ABB RobotStudio station: sesion6_EstacionDePartidaSoloRobotFin.rspag

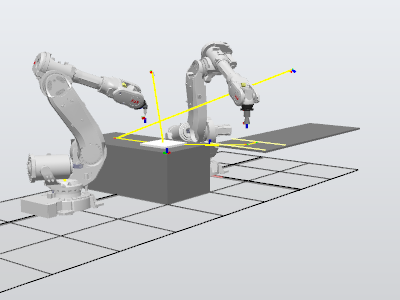
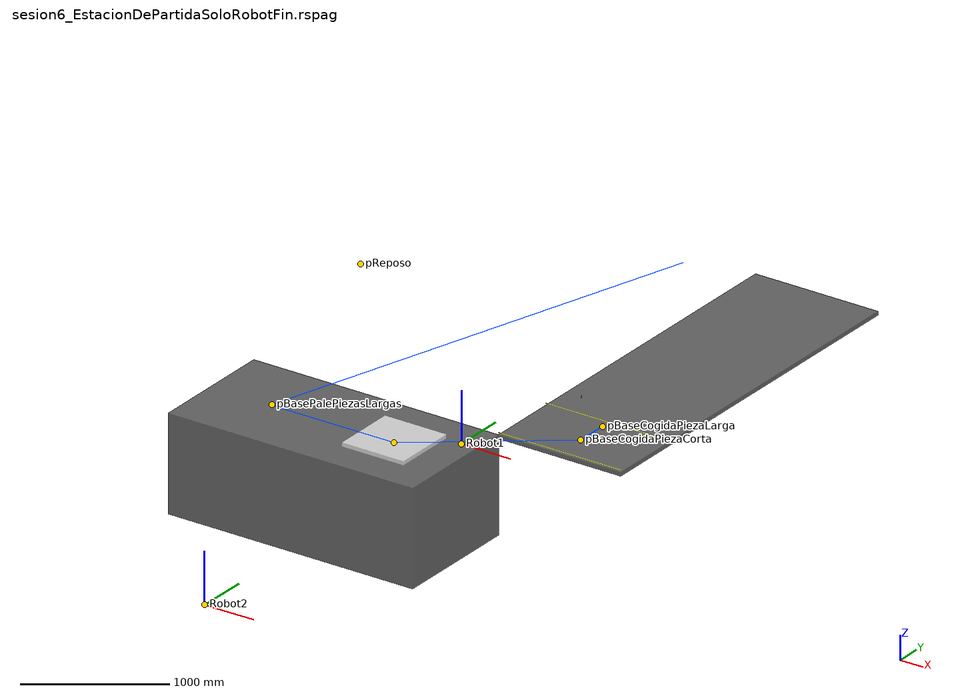
[picture v1: parts stored in the station drawn from their meshes, with robot base, taught points and paths (robot models come from the ABB library and are not in the file)]
--- station ---
Station sesion7_EstacionDePartida_1 (saved by RobotStudio 24.1.10713.1)
Controller Controlador3, task T_ROB1: task frame (RAPID world) sits at (0, -3000, 0) mm, rotated rx 0 ry 0 rz 90 deg in the station
Controller Sistema6
  mechanical unit ROB_1: Robot1, 6 joints, base frame (0, 0, 0) mm
Controller Controlador3
  mechanical unit ROB_1: Robot2, 6 joints, base frame (0, 0, 0) mm
Layout (positions relative to the parent item):
  - Ventosa [mechanism] at (1500, -750, 1280) mm, rotated rx -180 ry 0 rz -180 deg
      TCP Ventosa at (0, 0, 200) mm
      links: PiezaVentosa
  - Robot1 [mechanism, from %ABB.RobotStudio.Models.IRB6640%\IRB6640_180_255_G_04.rslib] at (0, 0, 0) mm; joint values [-0.4636, 0.2346, 0.2413, 0, 1.095, -0.4636] (rad or m)
  - CI_VentosaVacuostato [smart component]
      signals: DI ActivaVentosa, DO Vacuostato
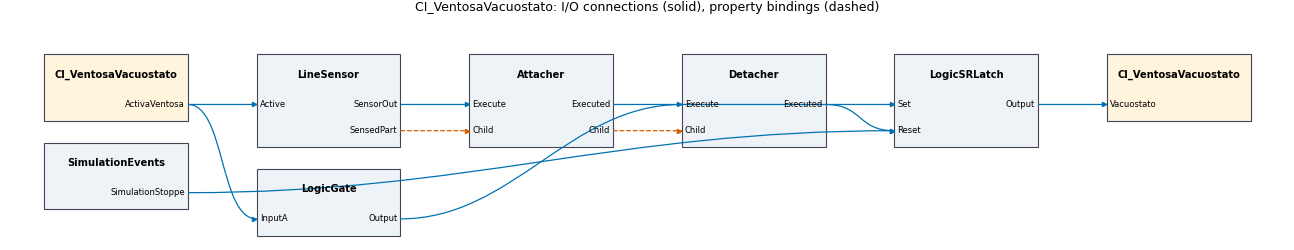
      connections:
        CI_VentosaVacuostato.ActivaVentosa -> LineSensor.Active
        LineSensor.SensorOut -> Attacher.Execute
        Attacher.Executed -> LogicSRLatch.Set
        LogicSRLatch.Output -> CI_VentosaVacuostato.Vacuostato
        Detacher.Executed -> LogicSRLatch.Reset
        SimulationEvents.SimulationStopped -> LogicSRLatch.Reset
        CI_VentosaVacuostato.ActivaVentosa -> LogicGate.InputA
        LogicGate.Output -> Detacher.Execute
        LineSensor.SensedPart => Attacher.Child
        Attacher.Child => Detacher.Child
    - LineSensor [smart component, from Components\LineSensor.rslib] at (1500, -750, 1080) mm, rotated rx -180 ry 0 rz -180 deg
        properties: Start=[0 0 -0.002]; End=[0 0 0.02]; Radius=0.002; SensedPart=(none); SensedPoint=[0.5 -1.49999987792969 0.780095153808594]; Length=0.022; Tag=(none)
      - _sensorPart_ [part], size 4 x 4 x 22 mm
    - SimulationEvents [smart component, from Components\SimulationEvents.rslib]
    - LogicSRLatch [smart component, from Components\LogicSRLatch.rslib]
    - Attacher [smart component, from Components\Attacher.rslib]
        properties: Parent=Ventosa; Flange=0; Child=(none); Mount=false; Offset=[0 0 0]; Orientation=[0 0 0]
    - Detacher [smart component, from Components\Detacher.rslib]
        properties: Child=(none); KeepPosition=true
    - LogicGate [smart component, from Components\LogicGate.rslib]
        properties: Operator=NOT; Delay=0.1
  - MesaPaletizadoParteIzq [part], size 1000 x 1000 x 750 mm
  - MesaPaletizadoParteDer [part], size 1000 x 1000 x 750 mm
  - cintaTransportadora [part], size 1000 x 3000 x 30 mm
  - PiezaLarga [part], size 500 x 1000 x 30 mm
  - PiezaCorta [part], size 500 x 500 x 30 mm
  - CI_SensoresCinta [smart component]
      signals: DI ActivaSensores, DO FinalCintaDetectado, DO PiezaLargaDetectada
      connections:
        CI_SensoresCinta.ActivaSensores -> LineSensorFinalCinta.Active
        CI_SensoresCinta.ActivaSensores -> LineSensorPiezaLarga.Active
        LineSensorPiezaLarga.SensorOut -> CI_SensoresCinta.PiezaLargaDetectada
        LineSensorFinalCinta.SensorOut -> CI_SensoresCinta.FinalCintaDetectado
    - LineSensorFinalCinta [smart component, from Components\LineSensor.rslib]
        properties: Start=[1 -1 0.765]; End=[2 -1 0.765]; Length=1; Radius=0.002; Tag=(none); SensedPart=(none); SensedPoint=[0 0 0]
      - _sensorPart_ [part], size 1000 x 4 x 4 mm
    - LineSensorPiezaLarga [smart component, from Components\LineSensor.rslib]
        properties: Start=[1 -0.45 0.765]; End=[2 -0.45 0.765]; Length=1; Radius=0.002; Tag=(none); SensedPart=(none); SensedPoint=[0 0 0]
      - _sensorPart_ [part], size 1000 x 4 x 4 mm
  - CI_CintaTransportadora [smart component]
      signals: DI PideNuevaPieza, DI MueveCinta, DI Desencolar
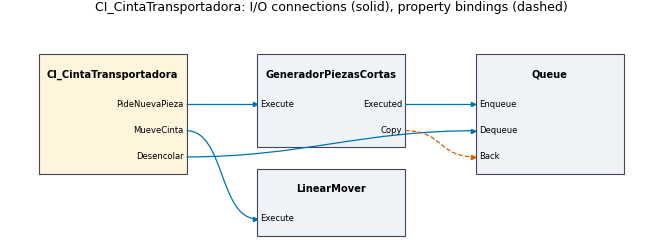
      connections:
        GeneradorPiezasCortas.Executed -> Queue.Enqueue
        CI_CintaTransportadora.PideNuevaPieza -> GeneradorPiezasCortas.Execute
        CI_CintaTransportadora.MueveCinta -> LinearMover.Execute
        CI_CintaTransportadora.Desencolar -> Queue.Dequeue
        GeneradorPiezasCortas.Copy => Queue.Back
    - GeneradorPiezasCortas [smart component, from Components\Source.rslib]
        properties: Source=PiezaCorta; Copy=(none); Parent=(none); Position=[1.25 1.5 0.75]; Orientation=[0 0 0]; Transient=false; PhysicsBehavior=-1
    - LinearMover [smart component, from Components\LinearMover.rslib]
        properties: Object=Queue; Direction=[0 -0.001 0]; Speed=0.2; Reference=Global; ReferenceObject=(none)
    - Queue [smart component, from Components\Queue.rslib]
        properties: Back=(none); Front=(none); Queue={d6de95e9-a5e4-462f-8fb5-12ca184cec83}; NumberOfObjects=0
  - PiezaCorta_5 [part] at (249.2, -1250, 750) mm, rotated rx 0 ry 0 rz -90 deg, size 500 x 500 x 30 mm
  - Robot2 [mechanism, from %ABB.RobotStudio.Models.IRB6640%\IRB6640_180_255_G_04.rslib] at (0, -3000, 0) mm, rotated rx 0 ry 0 rz 90 deg; joint values [-0.5264, -0.4516, 0.7886, 0.4989, 0.7029, -0.8234] (rad or m)
  - MyTool [mechanism, from Training Objects\myTool.rslib] at (500, -2016.33, 1400.53) mm, rotated rx 180 ry 38 rz -90 deg
Attachment: Ventosa is attached to Robot1 / Link6
Attachment: LineSensor is attached to Ventosa / PiezaVentosa
Attachment: MyTool is attached to Robot2 / Link6
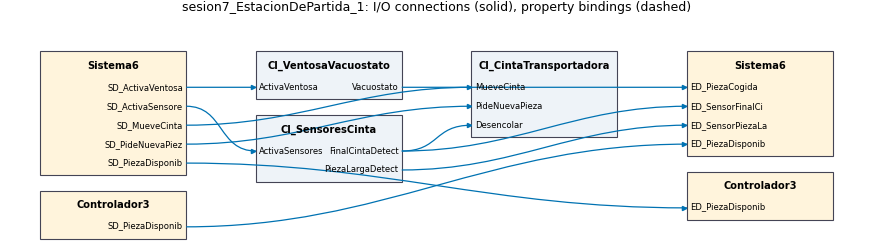
Station logic (signal -> signal, property => property):
  CI_VentosaVacuostato.Vacuostato -> Sistema6.ED_PiezaCogida
  Sistema6.SD_ActivaVentosa -> CI_VentosaVacuostato.ActivaVentosa
  CI_SensoresCinta.FinalCintaDetectado -> Sistema6.ED_SensorFinalCinta
  CI_SensoresCinta.PiezaLargaDetectada -> Sistema6.ED_SensorPiezaLarga
  Sistema6.SD_ActivaSensores -> CI_SensoresCinta.ActivaSensores
  Sistema6.SD_MueveCinta -> CI_CintaTransportadora.MueveCinta
  Sistema6.SD_PideNuevaPieza -> CI_CintaTransportadora.PideNuevaPieza
  CI_SensoresCinta.FinalCintaDetectado -> CI_CintaTransportadora.Desencolar
  Sistema6.SD_PiezaDisponible -> Controlador3.ED_PiezaDisponible
  Controlador3.SD_PiezaDisponibleAck -> Sistema6.ED_PiezaDisponibleAck

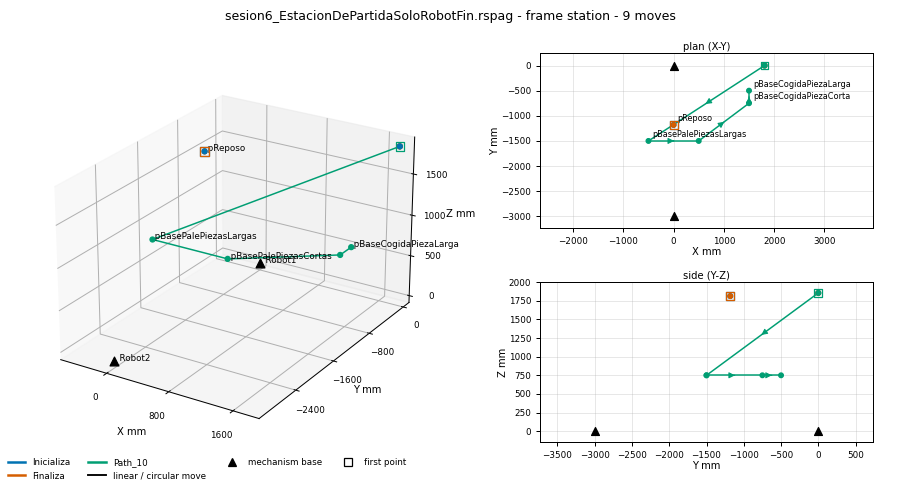
[picture p0: tool path of sesion6_EstacionDePartidaSoloRobotFin.rspag in frame station, 9 of 20 moves have a stored position in this frame; points joined in program order, loops and branches not executed]
--- Backups/Controlador3/RAPID/TASK1/PROGMOD/CalibData.mod ---
MODULE CalibData
    PERS tooldata MyTool:=[TRUE,[[31.792631019,0,229.638935148],[0.945518576,0,0.325568154,0]],[1,[0,0,1],[1,0,0,0],0,0,0]];
    TASK PERS wobjdata WO_Paletizado:=[FALSE,TRUE,"",[[1000,-1000,750],[1,0,0,0]],[[0,0,0],[1,0,0,0]]];
ENDMODULE

--- Backups/Controlador3/RAPID/TASK1/PROGMOD/Module1.mod ---
MODULE Module1
        CONST robtarget pReposo:=[[1818.681916784,0,1812.64730631],[0.190808996,0,0.981627183,0],[0,0,0,0],[9E+09,9E+09,9E+09,9E+09,9E+09,9E+09]];
    CONST robtarget pBasePalePiezasCortas:=[[500,500,0],[0,0,1,0],[-1,0,0,0],[9E+09,9E+09,9E+09,9E+09,9E+09,9E+09]];
    CONST robtarget pBasePalePiezasLargas:=[[500,1500,0],[0,0,1,0],[0,-1,0,0],[9E+09,9E+09,9E+09,9E+09,9E+09,9E+09]];
    PROC Inicializa ()
      MoveJ pReposo, v3000, fine, MyTool;
      Reset SD_PiezaDisponibleAck;
   ENDPROC
   PROC Finaliza ()
      MoveJ pReposo, v3000, fine, MyTool;
      Reset SD_PiezaDisponibleAck;
   ENDPROC
      PROC Main ()
      VAR num nPiezas;

      Inicializa;

      FOR nPiezas FROM 1 TO 20 DO
         WaitDI ED_PiezaDisponible, 1;
         SetDO SD_PiezaDisponibleAck, 1;
         WaitTime 0.3;
         Reset SD_PiezaDisponibleAck;
         TaladraPieza pBasePalePiezasCortas, nPiezas, 30;
      ENDFOR

      Finaliza;
   ENDPROC
      PROC TaladraPieza (robtarget pBase, num nPiezas, num altoPieza)
      VAR robtarget pTaladrado;
      VAR robtarget pAprox;
      VAR robtarget pEspera;
      VAR num distSeguridadZ := 300;
      VAR num distSeguridadEsperaX := -400;


      pTaladrado := Offs (pBasePalePiezasCortas, 0, 0, altoPieza*nPiezas);
      pAprox := Offs (pTaladrado, 0, 0, distSeguridadZ);
      pEspera := Offs (pTaladrado, distSeguridadEsperaX, 0, distSeguridadZ);

      MoveJ pAprox, v3000, z100, MyTool, \WObj:=WO_Paletizado;
      MoveL pTaladrado, v1000, fine, MyTool, \WObj:=WO_Paletizado;
      ! Aquí accionaríamos taladro. Simulamos con espera de 0.3 segundos:
      WaitTime 0.3;
      MoveL pAprox, v1000, z100, MyTool, \WObj:=WO_Paletizado;
      MoveJ pEspera, v3000, z100, MyTool, \WObj:=WO_Paletizado;
   ENDPROC
ENDMODULE

--- Backups/Sistema6/RAPID/TASK1/PROGMOD/CalibData.mod ---
MODULE CalibData
	PERS tooldata Ventosa:=[TRUE,[[0,0,200],[1,0,0,0]],[1,[0,0,125],[1,0,0,0],0.002,0.002,0.0013]];
    TASK PERS wobjdata WO_Paletizado:=[FALSE,TRUE,"",[[1000,-2000,750],[0.707106781,0,0,0.707106781]],[[0,0,0],[1,0,0,0]]];
    TASK PERS wobjdata WO_CintaTransportadora:=[FALSE,TRUE,"",[[1000,-1000,750],[1,0,0,0]],[[0,0,0],[1,0,0,0]]];
ENDMODULE

--- Backups/Sistema6/RAPID/TASK1/PROGMOD/Module1.mod ---
MODULE Module1
    CONST robtarget pReposo:=[[1808.910161514,0,1855],[0.5,0,0.866025404,0],[0,0,0,0],[9E+09,9E+09,9E+09,9E+09,9E+09,9E+09]];
    CONST robtarget pBasePalePiezasLargas:=[[500,1500,0],[0,1,0,0],[-2,0,-1,0],[9E+09,9E+09,9E+09,9E+09,9E+09,9E+09]];
    CONST robtarget pBasePalePiezasCortas:=[[500,500,0],[0,1,0,0],[-1,0,0,0],[9E+09,9E+09,9E+09,9E+09,9E+09,9E+09]];
    CONST robtarget pBaseCogidaPiezaCorta:=[[500,250,0],[0,0,1,0],[-1,0,-1,0],[9E+09,9E+09,9E+09,9E+09,9E+09,9E+09]];
    CONST robtarget pBaseCogidaPiezaLarga:=[[500,500,0],[0,0,1,0],[-1,0,-1,0],[9E+09,9E+09,9E+09,9E+09,9E+09,9E+09]];
 PROC Inicializa ()
      MoveJ pReposo, v3000, fine, Ventosa, \WObj:=wobj0;
      Reset SD_ActivaVentosa;
      SetDO SD_ActivaSensores, 1;
      SetDO SD_MueveCinta, 1;
      Reset SD_PideNuevaPieza;
      Reset SD_PiezaDisponible;
   ENDPROC

   PROC Finaliza ()
      MoveJ pReposo, v3000, fine, Ventosa, \WObj:=wobj0;
      Reset SD_ActivaVentosa;
      Reset SD_PideNuevaPieza;
      Reset SD_MueveCinta;
      Reset SD_ActivaSensores;
      Reset SD_ActivaSensores;
      Reset SD_PiezaDisponible;
   ENDPROC

   PROC Main ()
      CONST num altoPieza := 30;
      VAR num nPiezas;

      Inicializa;

      FOR nPiezas FROM 1 TO 20 DO
         WaitDI ED_SensorFinalCinta, 1;
         LlevaPiezaAPale nPiezas, altoPieza;
         SetDO SD_PiezaDisponible, 1;
         WaitDI ED_PiezaDisponibleAck, 1;
         Reset SD_PiezaDisponible;
      ENDFOR

      Finaliza;
   ENDPROC

   PROC LlevaPiezaAPale (num nPiezas, num altoPieza)
      VAR robtarget pCoger;
      VAR robtarget pSoltar;
      VAR robtarget pCogerAprox;
      VAR robtarget pSoltarAprox;
      VAR num distSeguridad := 300;

      pCoger  := Offs (pBaseCogidaPiezaCorta, 0, 0, altoPieza);
      pSoltar := Offs (pBasePalePiezasCortas, 0, 0, altoPieza*nPiezas);

      pCogerAprox  := Offs (pCoger,  0, 0, distSeguridad);
      pSoltarAprox := Offs (pSoltar, 0, 0, distSeguridad);

      MoveJ pCogerAprox, v3000, z100, Ventosa, \WObj:=WO_CintaTransportadora;
      MoveLDO pCoger, v1000, fine, Ventosa, \WObj:=WO_CintaTransportadora, SD_ActivaVentosa, 1;
      WaitDI ED_PiezaCogida, 1;
      MoveL pCogerAprox, v1000, z100, Ventosa, \WObj:=WO_CintaTransportadora;
      MoveJ pSoltarAprox, v3000, z100, Ventosa, \WObj:=WO_Paletizado;
      MoveLDO pSoltar, v1000, fine, Ventosa, \WObj:=WO_Paletizado, SD_ActivaVentosa, 0;
      WaitDI ED_PiezaCogida, 0;
      MoveL pSoltarAprox, v1000, z100, Ventosa, \WObj:=WO_Paletizado;
      MoveJ pCogerAprox, v3000, z100, Ventosa, \WObj:=WO_CintaTransportadora;
   ENDPROC
    PROC Path_10()
        MoveL pReposo,v1000,z100,Ventosa\WObj:=wobj0;
        MoveL pBasePalePiezasLargas,v1000,z100,Ventosa\WObj:=WO_Paletizado;
        MoveL pBasePalePiezasCortas,v1000,z100,Ventosa\WObj:=WO_Paletizado;
        MoveL pBaseCogidaPiezaCorta,v1000,z100,Ventosa\WObj:=WO_CintaTransportadora;
        MoveL pBaseCogidaPiezaLarga,v1000,z100,Ventosa\WObj:=WO_CintaTransportadora;
    ENDPROC
ENDMODULE

--- Backups/Sistema6/RAPID/TASK1/SYSMOD/LINKEDM.sys ---
%%%
  VERSION:1
  LANGUAGE:ENGLISH
%%%

MODULE LINKEDM (SYSMODULE)

! FOLLOWER
!     Name of electronically linked follower axis used by operator at teach pendent.
      PERS string l_f_axis_name{5}       :=  ["",  "", "", "", ""];

!     Name of the mechanical unit for follower axis.
      PERS string l_f_mecunt_n{5}  :=  ["", "", "", "", ""];

!     Linked follower axis number in the mechanical unit (first axis in mech. unit is number 1).
      PERS num l_f_axis_no{5}      :=  [0,          0,   0,  0,  0];

! MASTER
!     Name of the mechanical unit for linked master axis.
      PERS string l_m_mecunt_n{5} :=  ["", "", "", "", ""];

!     Linked master axis number in the mechanical unit (first axis in mech. unit is number 1).
!     See axis number table in documentation for different master mechanical units.
      PERS num l_m_axis_no{5}     :=  [0,  0,  0,  0,  0];

! POSITION OFFSET
!     The increase of the allowed offset position between the master and follower
!     positions, used when starting AUTO mode. As soon as the offset is decreased
!     the old configurated parameter is used.
!     Example: 3 => the configurated value of allowed offset is increased 3 times.
      PERS num offset_ratio{5}       :=  [10,  10,   10,  10,  10];

! SPEED RATIO
!     Speed_ratio used in AUTO and JOG modes [ very_slow   slow    normal    fast]
!     Value 1 = max allowed manual speed.
      CONST num speed_ratio {20}      := [0.01, 0.01, 0.01, 0.01, 0.01,
                                          0.05, 0.05, 0.05, 0.05, 0.05,
                                          0.20, 0.20, 0.20, 0.20, 0.20,
                                          1.00, 1.00, 1.00, 1.00, 1.00];

! STEP SIZE
!     Displacement position used in JOG mode for each activation of positive or
!     negative movement.                  [very_short    short   normal   long]
!     Unit degees or meter.
      CONST num displacement {20}     := [0.001, 0.001, 0.001, 0.001, 0.001,
                                          0.005, 0.005, 0.005, 0.005, 0.005,
                                          0.020, 0.020, 0.020, 0.020, 0.020,
                                          0.100, 0.100, 0.100, 0.100, 0.100];


!-------------------------------------------------------------
 PROC Linked_m ()
      Linked_m_exe ;
 ENDPROC
ENDMODULE

--- Backups/Controlador3/SYSPAR/EIO.cfg ---
EIO:CFG_1.0:6:1::
#
INDUSTRIAL_NETWORK:

      -Name "DeviceNet" -Label "DeviceNet Master/Slave Network" -Address "2"
#
DEVICENET_DEVICE:

      -Name "MiDeviceNet"
#
DEVICENET_INTERNAL_DEVICE:

      -Name "DN_Internal_Device" -VendorName "ABB Robotics"\
      -ProductName "DeviceNet Internal Slave Device"
#
EIO_SIGNAL:

      -Name "ED_PiezaDisponible" -SignalType "DI" -Device "MiDeviceNet"\
      -Label "ED_PiezaDisponible" -DeviceMap "0"

      -Name "SD_PiezaDisponibleAck" -SignalType "DO" -Device "MiDeviceNet"\
      -Label "SD_PiezaDisponibleAck" -DeviceMap "0"

--- Backups/Sistema6/SYSPAR/EIO.cfg ---
EIO:CFG_1.0:6:1::
#
INDUSTRIAL_NETWORK:

      -Name "DeviceNet" -Label "DeviceNet Master/Slave Network" -Address "2"
#
DEVICENET_DEVICE:

      -Name "MiDeviceNet" -Label "MiDeviceNet"
#
DEVICENET_INTERNAL_DEVICE:

      -Name "DN_Internal_Device" -VendorName "ABB Robotics"\
      -ProductName "DeviceNet Internal Slave Device"
#
EIO_SIGNAL:

      -Name "ED_PiezaCogida" -SignalType "DI" -Device "MiDeviceNet"\
      -Label "ED_PiezaCogida" -DeviceMap "0" -Access "All"

      -Name "SD_ActivaVentosa" -SignalType "DO" -Device "MiDeviceNet"\
      -Label "SD_ActivaVentosa" -DeviceMap "0" -Access "All"

      -Name "ED_SensorFinalCinta" -SignalType "DI" -Device "MiDeviceNet"\
      -Label "ED_SensorFinalCinta" -DeviceMap "1" -Access "All"

      -Name "ED_SensorPiezaLarga" -SignalType "DI" -Device "MiDeviceNet"\
      -Label "ED_SensorPiezaLarga" -DeviceMap "2" -Access "All"

      -Name "SD_ActivaSensores" -SignalType "DO" -Device "MiDeviceNet"\
      -Label "SD_ActivaSensores" -DeviceMap "1" -Access "All"

      -Name "SD_MueveCinta" -SignalType "DO" -Device "MiDeviceNet"\
      -Label "SD_MueveCinta" -DeviceMap "2" -Access "All"

      -Name "SD_PideNuevaPieza" -SignalType "DO" -Device "MiDeviceNet"\
      -Label "SD_PideNuevaPieza" -DeviceMap "3" -Access "All"

      -Name "SD_PiezaDisponible" -SignalType "DO" -Device "MiDeviceNet"\
      -Label "SD_PiezaDisponible" -DeviceMap "4"

      -Name "ED_PiezaDisponibleAck" -SignalType "DI" -Device "MiDeviceNet"\
      -Label "ED_PiezaDisponibleAck" -DeviceMap "3"
